TYPE csp_transfer_accumulator_belt_status_enum :
(
	CSP_TRANSFER_ACCUMULATOR_BELT_STATUS_NOT_INITIALIZED 							:=  0,
	CSP_TRANSFER_ACCUMULATOR_BELT_STATUS_DISABLED 									:=  10,
	CSP_TRANSFER_ACCUMULATOR_BELT_STATUS_ENABLE_REQUEST 							:=  20,
	CSP_TRANSFER_ACCUMULATOR_BELT_STATUS_ENABLING 									:=  30,
	CSP_TRANSFER_ACCUMULATOR_BELT_STATUS_ENABLED 									:=  40,
	CSP_TRANSFER_ACCUMULATOR_BELT_STATUS_HOME_REQUEST								:=  50,
	CSP_TRANSFER_ACCUMULATOR_BELT_STATUS_HOMING									:=  60,
	CSP_TRANSFER_ACCUMULATOR_BELT_STATUS_HOME_DONE									:=  70,
	CSP_TRANSFER_ACCUMULATOR_BELT_STATUS_CALCULATING_SLAVE_POSITION				:=  90,
	CSP_TRANSFER_ACCUMULATOR_BELT_STATUS_WAITING_SLAVE_ENGAGE						:= 100,
	CSP_TRANSFER_ACCUMULATOR_BELT_STATUS_PHASE_REQUEST								:= 140,
	CSP_TRANSFER_ACCUMULATOR_BELT_STATUS_PHASING									:= 150,
	CSP_TRANSFER_ACCUMULATOR_BELT_STATUS_PHASED									:= 160,
	CSP_TRANSFER_ACCUMULATOR_BELT_STATUS_CAM_ENGAGED_REQ							:= 170,
	CSP_TRANSFER_ACCUMULATOR_BELT_STATUS_AXIS_ENGAGE_VERIFY						:= 180,
	CSP_TRANSFER_ACCUMULATOR_BELT_STATUS_CAM_ENGAGED_EXTEND								:= 190,
	CSP_TRANSFER_ACCUMULATOR_BELT_STATUS_CAM_DISENAGE_WAIT							:= 191,
	CSP_TRANSFER_ACCUMULATOR_BELT_STATUS_CAM_ENGAGED_RETRACT							:= 192,
	CSP_TRANSFER_ACCUMULATOR_BELT_STATUS_CAM_TABLE_READ							:= 195,
	CSP_TRANSFER_ACCUMULATOR_BELT_STATUS_CALCULATE_SLAVE_POSITION_REQUEST			:= 196,
	CSP_TRANSFER_ACCUMULATOR_BELT_STATUS_READY										:= 197,
	CSP_TRANSFER_ACCUMULATOR_BELT_STATUS_RUNNING									:= 200,
	CSP_TRANSFER_ACCUMULATOR_BELT_STATUS_MOVING									:= 205,
	CSP_TRANSFER_ACCUMULATOR_BELT_STATUS_DISENGAGE_REQUEST						:= 210,
	CSP_TRANSFER_ACCUMULATOR_BELT_STATUS_DISENGAGING								:= 211,	
	CSP_TRANSFER_ACCUMULATOR_BELT_STATUS_REJECT									:= 220,
	CSP_TRANSFER_ACCUMULATOR_BELT_STATUS_REJECT_WAITING							:= 221,
	CSP_TRANSFER_ACCUMULATOR_BELT_STATUS_REJECT_COMPLETE							:= 222,
	CSP_TRANSFER_ACCUMULATOR_BELT_STATUS_STOP_REQUEST 								:= 500,
	CSP_TRANSFER_ACCUMULATOR_BELT_STATUS_DISABLE_REQUEST 							:= 530,
	CSP_TRANSFER_ACCUMULATOR_BELT_STATUS_DISABLING 								:= 540
) := CSP_TRANSFER_ACCUMULATOR_BELT_STATUS_NOT_INITIALIZED;
END_TYPE

(* stored: Version 1.1.0.1, ProductVersion 3.1.4022.12
   DUT csp_transfer_accumulator_belt_status_enum: Id {e5cbc954-2d91-4e11-b15f-d420bc9b00a6} *)
